(* CoDeSys 2.3.9.28 project: AULA05_EX01.pro *)
(* Libraries: Standard.lib 27.1.09 11:27:38, Util.lib 27.1.09 11:27:38, IecSfc.lib*24.11.08 08:07:15, SysLibTime.lib*27.1.09 11:27:38, SysTaskInfo.lib 24.11.08 08:07:15, SYSLIBCALLBACK.LIB 27.1.09 11:27:38 *)

(* PLC configuration (modules and I/O channels)
Hexswitch AT %IB0 [HexSwitch] rotary switch 0 = STOP, 1-15 = RUN
IOModules [CPX_MASTER] node 0, in %IB4 out %QB0
  8DI/8DO [CPX-8DI_8DO_Multi_I_O_module_1] node 0, in %IB4 out %QB0 {StringParam = 4,8,1,8,1; ByteParam = 7; ByteParam = 81; ByteParam = 0; ByteParam = 0; ByteParam = 0; ByteParam = 0; ByteParam = 0; IdleStateParam = 0; IdleModeParam = 255; IdleStateParam = 0; IdleModeParam = 255; IdleStateParam = 0; IdleModeParam = 255; IdleStateParam = 0; IdleModeParam = 255}
    AT %IB4 [ByteInput] -
    AT %QB0 [ByteOutput] -
  8DI/8DO [CPX-8DI_8DO_Multi_I_O_module_1] node 1, in %IB8 out %QB4 {StringParam = 4,8,1,8,1; ByteParam = 7; ByteParam = 81; ByteParam = 0; ByteParam = 0; ByteParam = 0; ByteParam = 0; ByteParam = 0; IdleStateParam = 0; IdleModeParam = 255; IdleStateParam = 0; IdleModeParam = 255; IdleStateParam = 0; IdleModeParam = 255; IdleStateParam = 0; IdleModeParam = 255}
    AT %IB8 [ByteInput] -
    AT %QB4 [ByteOutput] -
*)

(* Global variable list: Global_Variables *)
VAR_GLOBAL

	START AT %IX2.0 : BOOL;
	STOP AT %IX2.1 : BOOL;
	B1 AT %IX2.2 : BOOL;
	S1 AT %IX2.3 : BOOL;
	S2 AT %IX2.4 : BOOL;

	M1 AT %QX0.0 : BOOL;
	Y1 AT %QX0.1 : BOOL;
	Y2 AT %QX0.2 : BOOL;
	M2 AT %QX0.3 : BOOL;

END_VAR

(* POU PLC_PRG, LD *)
PROGRAM PLC_PRG
VAR
END_VAR
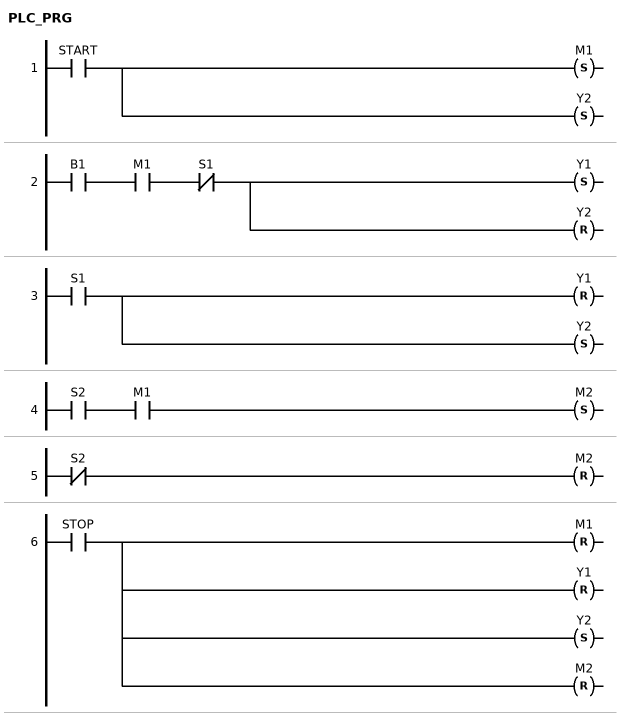
_LD_ (* Ladder Diagram *)
NETWORK 1
	[START] --- (S M1) (S Y2)
NETWORK 2
	[B1] - [M1] - [/S1] --- (S Y1) (R Y2)
NETWORK 3
	[S1] --- (R Y1) (S Y2)
NETWORK 4
	[S2] - [M1] --- (S M2)
NETWORK 5
	[/S2] --- (R M2)
NETWORK 6
	[STOP] --- (R M1) (R Y1) (S Y2) (R M2)
_END_LD_
(* the same logic as Structured Text *)
(* Network 1 *)
IF START THEN M1 := TRUE; Y2 := TRUE; END_IF;
(* Network 2 *)
IF B1 AND M1 AND NOT S1 THEN Y1 := TRUE; Y2 := FALSE; END_IF;
(* Network 3 *)
IF S1 THEN Y1 := FALSE; Y2 := TRUE; END_IF;
(* Network 4 *)
IF S2 AND M1 THEN M2 := TRUE; END_IF;
(* Network 5 *)
IF NOT S2 THEN M2 := FALSE; END_IF;
(* Network 6 *)
IF STOP THEN M1 := FALSE; Y1 := FALSE; Y2 := TRUE; M2 := FALSE; END_IF;
END_PROGRAM
